Fanuc KAREL source: kt00700.KL

-- PROVISIONAL review KL for V940-1; original PC SHA256 7dcf3b258d4183cb8ed154e9398aa868fdd8813b084ad5d079b8aa38b45921a9
-- Incomplete behavior may be omitted. Consult companion uncertainty JSON. Do not deploy.
PROGRAM KT00700
%NOLOCKGROUP
VAR
  OUT : INTEGER
-- UNRESOLVED_DECL C1 type=00001c
-- UNRESOLVED_DECL C2 type=00001c
BEGIN
  -- V9_ZERO_TABLE_METADATA_HINT layout=0001; no indexed target words; source/name/runtime held
  -- UNRESOLVED_PC offsets 5-15; opcodes 9D,22,A5
  -- UNRESOLVED_PC offsets 20-30; opcodes 9C,22,A5
  -- UNRESOLVED_PC offsets 35-45; opcodes 9D,22,A5
  -- UNRESOLVED_PC offsets 50-60; opcodes 9C,22,A5
  -- UNRESOLVED_PC offsets 65-77; opcodes 21,23
  -- UNRESOLVED_PC offsets 82-86; opcodes 7F
END KT00700
